FUNCTION INTERNAL Tc2MC2_TO_Tco_JogMode : BOOL
VAR_INPUT
    Tc2MC2JogMode : Tc2_MC2.E_JogMode;
END_VAR
VAR_IN_OUT
    TcoJogMode : eJogMode;
END_VAR

CASE Tc2MC2JogMode OF
    Tc2_MC2.MC_JOGMODE_STANDARD_SLOW:
        TcoJogMode := eJogMode.MC_JOGMODE_STANDARD_SLOW;
        Tc2MC2_TO_Tco_JogMode := TRUE;
    Tc2_MC2.MC_JOGMODE_STANDARD_FAST:
        TcoJogMode := eJogMode.MC_JOGMODE_STANDARD_FAST;
        Tc2MC2_TO_Tco_JogMode := TRUE;
    Tc2_MC2.MC_JOGMODE_CONTINOUS:
        TcoJogMode := eJogMode.MC_JOGMODE_CONTINOUS;
        Tc2MC2_TO_Tco_JogMode := TRUE;
    Tc2_MC2.MC_JOGMODE_INCHING:
        TcoJogMode := eJogMode.MC_JOGMODE_INCHING;
        Tc2MC2_TO_Tco_JogMode := TRUE;
    Tc2_MC2.MC_JOGMODE_INCHING_MODULO:
        TcoJogMode := eJogMode.MC_JOGMODE_INCHING_MODULO;
        Tc2MC2_TO_Tco_JogMode := TRUE;
ELSE
    Tc2MC2_TO_Tco_JogMode := FALSE;
END_CASE

END_FUNCTION

(* stored: Version 1.1.0.1, ProductVersion 3.1.4024.9
   POU Tc2MC2_TO_Tco_JogMode: Id {beaf1796-310e-0ab2-3315-a0a70ac7f3db}, SpecialFunc None *)
